# EPICS substitutions: rtApp/Db/tmicro_block.substitutions
file tmicro_block.template {
    pattern{M,B}
    {0,0}
    {0,1}
    {0,2}
    {0,3}
    {0,4}
    {0,5}
    {0,6}
    {0,7}
    {1,0}
    {1,1}
    {1,2}
    {1,3}
    {1,4}
    {1,5}
    {1,6}
    {1,7}
    {2,0}
    {2,1}
    {2,2}
    {2,3}
    {2,4}
    {2,5}
    {2,6}
    {2,7}
}
